// TwinCAT 3 PLC project PLC
// ProgramVersion: 3.1.4026.21
// libraries:
//   mobject-core, * (mobject)
//   Tc2_Standard, * (Beckhoff Automation GmbH)
//   Tc2_System, * (Beckhoff Automation GmbH)
//   Tc2_Utilities, * (Beckhoff Automation GmbH)
// project tree:
//   EL2574/DUT/ EL2574_IO.TcDUT, EL2574_Command.TcDUT, EL2574_IO_Control_Color.TcDUT, EL2574_IO_Status.TcDUT, EL2574_IO_Control.TcDUT
//   EL2574/ EL2574_CommandMode.TcPOU, HtmlColorCodeToRGBA.TcPOU, Section.TcDUT
//   EL2574/Interface/ I_EL2574_CommandMode.TcIO
//   / MAIN.TcPOU, PlcTask.TcTTO
// real-time tasks:
//   TASK PlcTask: cycle T#10ms, priority 20, ADS port 350
// I/O:
//   DEVICE CX (EtherCAT), AmsNetId 0.0.0.0.2.1
//     Term 1 (EK1200) [EK1200-5000 EtherCAT Power supply (2A E-Bus)]
//       LED 1-4 (EL2574) [EL2574 4 Ch. Pixel LED Controller]
//         modules: SlotGroup 1 (Slot 1, 2) (2xASYNC), SlotGroup 1 (Slot 1, 2) (2xASYNC), SlotGroup 2 (Slot 3, 4) (2xASYNC), SlotGroup 2 (Slot 3, 4) (2xASYNC)
//       LED 5-8 (EL2574) [EL2574 4 Ch. Pixel LED Controller]
//         modules: SlotGroup 1 (Slot 1, 2) (2xASYNC), SlotGroup 1 (Slot 1, 2) (2xASYNC), SlotGroup 2 (Slot 3, 4) (2xASYNC), SlotGroup 2 (Slot 3, 4) (2xASYNC)
// variable links:
//   (this object) <-> CX (EtherCAT)/Term 1 (EK1200)/LED 1-4 (EL2574)
//     PlcTask Inputs/MAIN.LED1.pdo.Status <-> SlotGroup 1 (Slot 1, 2) (2xASYNC)/Status Channel 1/Status
//     PlcTask Inputs/MAIN.LED2.pdo.Status <-> SlotGroup 1 (Slot 1, 2) (2xASYNC)/Status Channel 2/Status
//     PlcTask Inputs/MAIN.LED3.pdo.Status <-> SlotGroup 2 (Slot 3, 4) (2xASYNC)/Status Channel 1/Status
//     PlcTask Inputs/MAIN.LED4.pdo.Status <-> SlotGroup 2 (Slot 3, 4) (2xASYNC)/Status Channel 2/Status
//     PlcTask Outputs/MAIN.LED1.pdo.Control <-> SlotGroup 1 (Slot 1, 2) (2xASYNC)/Control Channel 1/Control
//     PlcTask Outputs/MAIN.LED2.pdo.Control <-> SlotGroup 1 (Slot 1, 2) (2xASYNC)/Control Channel 2/Control
//     PlcTask Outputs/MAIN.LED3.pdo.Control <-> SlotGroup 2 (Slot 3, 4) (2xASYNC)/Control Channel 1/Control
//     PlcTask Outputs/MAIN.LED4.pdo.Control <-> SlotGroup 2 (Slot 3, 4) (2xASYNC)/Control Channel 2/Control
//   (this object) <-> CX (EtherCAT)/Term 1 (EK1200)/LED 5-8 (EL2574)
//     PlcTask Inputs/MAIN.LED5.pdo.Status <-> SlotGroup 1 (Slot 1, 2) (2xASYNC)/Status Channel 1/Status
//     PlcTask Outputs/MAIN.LED5.pdo.Control <-> SlotGroup 1 (Slot 1, 2) (2xASYNC)/Control Channel 1/Control

CONFIGURATION PLC
    RESOURCE PLC ON TwinCAT3
        TASK PlcTask(INTERVAL := T#10ms, PRIORITY := 20);
        PROGRAM MAIN WITH PlcTask : MAIN;
    END_RESOURCE
END_CONFIGURATION

// ---- EL2574/DUT/EL2574_IO.TcDUT
TYPE EL2574_IO :
	STRUCT
		Status	AT %I* : EL2574_IO_Status;
		Control AT %Q* : EL2574_IO_Control;
	END_STRUCT
END_TYPE

// ---- EL2574/DUT/EL2574_Command.TcDUT
TYPE EL2574_Command :
	STRUCT
		Send	   : BOOL;
		Update	   : BOOL;
		Command	   : USINT;
		Index	   : UINT;
		Length	   : UINT;
		Parameter  : UINT;
		ColorRed   : USINT;
		ColorGreen : USINT;
		ColorBlue  : USINT;
		ColorWhite : USINT;
	END_STRUCT
END_TYPE

// ---- EL2574/DUT/EL2574_IO_Control_Color.TcDUT
TYPE EL2574_IO_Control_Color :
	STRUCT
		Red	  : USINT;
		Green : USINT;
		Blue  : USINT;
		White : USINT;
	END_STRUCT
END_TYPE

// ---- EL2574/DUT/EL2574_IO_Status.TcDUT
TYPE EL2574_IO_Status :
	STRUCT
		Busy					 : BIT;
		Transmit				 : BIT;
		Send_Acknowledge		 : BIT;
		Update_Acknowledge		 : BIT;
		Command_Acknowledge		 : BIT;
		Command_Reject			 : BIT;
		Warning					 : BIT;
		Error					 : BIT;
		Input_Cycle_Counter_Bit0 : BIT;
		Input_Cycle_Counter_Bit1 : BIT;
        {attribute 'hide'}
		_reserved1				 : BIT;
        {attribute 'hide'}
		_reserved2				 : BIT;
        {attribute 'hide'}
		_reserved3				 : BIT;
        {attribute 'hide'}
		_reserved4				 : BIT;
        {attribute 'hide'}
		_reserved5				 : BIT;
        {attribute 'hide'}
		_reserved6				 : BIT;
	END_STRUCT
END_TYPE

// ---- EL2574/DUT/EL2574_IO_Control.TcDUT
TYPE EL2574_IO_Control :
	STRUCT
		Execute : BIT;
		Send	: BIT;
		Update	: BIT;
		{attribute 'hide'}
		_reserved1 : BIT;
		{attribute 'hide'}
		_reserved2 : BIT;
		{attribute 'hide'}
		_reserved3 : BIT;
		{attribute 'hide'}
		_reserved4 : BIT;
		{attribute 'hide'}
		_reserved5 : BIT;
		Command	   : USINT;
		Index	   : UINT;
		Length	   : UINT;
		Parameter  : UINT;
		Color	   : EL2574_IO_Control_Color;
	END_STRUCT
END_TYPE

// ---- EL2574/Section.TcDUT
{attribute 'qualified_only'}
{attribute 'strict'}
{attribute 'to_string'}
TYPE Section : (
		None := 0,
		Accelerometer,
		Drives,
		Converter,
		Linux,
		Safety
	);
END_TYPE

// ---- EL2574/Interface/I_EL2574_CommandMode.TcIO
INTERFACE I_EL2574_CommandMode

METHOD PUBLIC ClearAll : I_EL2574_CommandMode
VAR_INPUT
END_VAR
END_METHOD

METHOD PUBLIC ColorGradient2Point : I_EL2574_CommandMode
VAR_INPUT
	StartPosition  : UINT;
	NumberOfPixels : UINT;
	Color1		   : STRING(9);
	Color2		   : STRING(9);
END_VAR
END_METHOD

METHOD PUBLIC ColorGradient3Point : I_EL2574_CommandMode
VAR_INPUT
	StartPosition  : UINT;
	NumberOfPixels : UINT;
	Color1		   : STRING(9);
	Color2		   : STRING(9);
	Color3		   : STRING(9);
END_VAR
END_METHOD

METHOD PUBLIC ColorGradient4Point : I_EL2574_CommandMode
VAR_INPUT
	StartPosition  : UINT;
	NumberOfPixels : UINT;
	Color1		   : STRING(9);
	Color2		   : STRING(9);
	Color3		   : STRING(9);
	Color4		   : STRING(9);
END_VAR
END_METHOD

METHOD PUBLIC CopyPixels : I_EL2574_CommandMode
VAR_INPUT
	StartPosition  : UINT;
	NumberOfPixels : UINT;
	TargetPosition : UINT;
END_VAR
END_METHOD

METHOD PUBLIC FillColor : I_EL2574_CommandMode
VAR_INPUT
	StartPosition  : UINT;
	NumberOfPixels : UINT;
	Red			   : USINT;
	Green		   : USINT;
	Blue		   : USINT;
	White		   : USINT;
END_VAR
END_METHOD

METHOD PUBLIC Invert : I_EL2574_CommandMode
VAR_INPUT
	StartPosition  : UINT;
	NumberOfPixels : UINT;
END_VAR
END_METHOD

METHOD PUBLIC MovePixels : I_EL2574_CommandMode
VAR_INPUT
	StartPosition  : UINT;
	NumberOfPixels : UINT;
	TargetPosition : UINT;
END_VAR
END_METHOD

METHOD PUBLIC RotateLeft : I_EL2574_CommandMode
VAR_INPUT
	StartPosition  : UINT;
	NumberOfPixels : UINT;
	Shift		   : UINT;
END_VAR
END_METHOD

METHOD PUBLIC RotateRight : I_EL2574_CommandMode
VAR_INPUT
	StartPosition  : UINT;
	NumberOfPixels : UINT;
	Shift		   : UINT;
END_VAR
END_METHOD

METHOD PUBLIC Send : I_EL2574_CommandMode
VAR_INPUT
END_VAR
END_METHOD

METHOD PUBLIC SendAndUpdate : I_EL2574_CommandMode
VAR_INPUT
END_VAR
END_METHOD

METHOD PUBLIC Update : I_EL2574_CommandMode
VAR_INPUT
END_VAR
END_METHOD

END_INTERFACE

// ---- MAIN.TcPOU
PROGRAM MAIN
VAR
	BackgroundColor		   : STRING(9) := '#fffafa';
	BackgroundColorRGB	   : ARRAY[0..3] OF USINT;
	DisplaySection		   : Section := Section.Linux;
	LED1				   : EL2574_CommandMode(10);
	LED2				   : EL2574_CommandMode(10);
	LED3				   : EL2574_CommandMode(10);
	LED4				   : EL2574_CommandMode(10);
	LED5				   : EL2574_CommandMode(10);
	onChange			   : r_Trig;
	previousDisplaySection : Section;
	State				   : (Idle,
		Clear,
		SetColor,
		SetColorUpdate);
	UpdateTon : TON;
	start	  : UINT;
	end		  : UINT;
END_VAR

VAR CONSTANT
	WHITE  : ARRAY[0..2] OF USINT := [255, 255, 255];
	RED	   : ARRAY[0..2] OF USINT := [255, 0, 0];
	BLUE   : ARRAY[0..2] OF USINT := [0, 0, 255];
	GREEN  : ARRAY[0..2] OF USINT := [0, 255, 0];
	YELLOW : ARRAY[0..2] OF USINT := [255, 255, 0];
END_VAR

BackgroundColorRGB := HtmlColorCodeToRGBA(BackgroundColor);
CASE State OF
	Idle:
		onChange(CLK := previousDisplaySection <> DisplaySection);
		IF OnChange.Q THEN
			PreviousDisplaySection := DisplaySection;
			LED1.ClearAll();
			LED2.ClearAll();
			LED3.ClearAll();
			LED4.FillColor(0,
						   75,
						   BackgroundColorRGB[0],
						   BackgroundColorRGB[1],
						   BackgroundColorRGB[2],
						   0);

			LED5.FillColor(0,
						   75,
						   BackgroundColorRGB[0],
						   BackgroundColorRGB[1],
						   BackgroundColorRGB[2],
						   0);

			State := Clear;
		END_IF

	Clear:
		UpdateTon(IN := TRUE, PT := T#100MS);
		IF UpdateTon.Q THEN
			UpdateTon(IN := FALSE);
			LED1.Update();
			LED2.Update();
			LED3.Update();
			LED4.Update();
			LED5.Update();
			State := SetColor;
		END_IF

	SetColor:
		CASE DisplaySection OF
			Section.None:
			Section.Accelerometer:
				LED2.FillColor(3,
							   3,
							   GREEN[0],
							   GREEN[1],
							   GREEN[2],
							   0);

			Section.Drives:
				LED1.FillColor(0,
							   100,
							   RED[0],
							   RED[1],
							   RED[2],
							   0);

				LED2.FillColor(0,
							   2,
							   RED[0],
							   RED[1],
							   RED[2],
							   0);

				LED3.ClearAll();

			Section.Linux:
				LED2.FillColor(4,
							   5,
							   WHITE[0],
							   WHITE[1],
							   WHITE[2],
							   0);

				LED3.ClearAll();

			Section.Safety:
				LED1.FillColor(0,
							   100,
							   YELLOW[0],
							   YELLOW[1],
							   YELLOW[2],
							   0);

				LED2.FillColor(0,
							   2,
							   YELLOW[0],
							   YELLOW[1],
							   YELLOW[2],
							   0);

				LED3.FillColor(0,
							   100,
							   YELLOW[0],
							   YELLOW[1],
							   YELLOW[2],
							   0);

			Section.Converter:
				LED2.FillColor(0,
							   2,
							   0,
							   0,
							   0,
							   0);

				LED2.FillColor(3,
							   3,
							   BLUE[0],
							   BLUE[1],
							   BLUE[2],
							   0);

				LED2.FillColor(4,
							   5,
							   0,
							   0,
							   0,
							   0);
		END_CASE

		State := SetColorUpdate;

	SetColorUpdate:
		UpdateTon(IN := TRUE, PT := T#100MS);
		IF UpdateTon.Q THEN
			UpdateTon(IN := FALSE);
			LED1.Update();
			LED2.Update();
			LED3.Update();
			LED4.Update();
			LED5.Update();
			State := IDLE;
		END_IF
END_CASE

LED1.CyclicCall();
LED2.CyclicCall();
LED3.CyclicCall();
LED4.CyclicCall();
LED5.CyclicCall();

END_PROGRAM

// ---- EL2574/EL2574_CommandMode.TcPOU
FUNCTION_BLOCK EL2574_CommandMode IMPLEMENTS I_EL2574_CommandMode
VAR
	totalPixels : UDINT;
	pdo			: EL2574_IO;
	commands	: Queue;
	errored		: BOOL;
END_VAR

VAR CONSTANT
	MAX_PIXELS			   : UDINT := 2048;
	COMMAND_NOP			   : USINT := 16#00;
	COMMAND_FILL		   : USINT := 16#01;
	COMMAND_CLEAR		   : USINT := 16#02;
	COMMAND_COPY		   : USINT := 16#03;
	COMMAND_MOVE		   : USINT := 16#04;
	COMMAND_ROTATE_LEFT	   : USINT := 16#05;
	COMMAND_ROTATE_RIGHT   : USINT := 16#06;
	COMMAND_REVERSE		   : USINT := 16#07;
	COMMAND_GRADIENT_START : USINT := 16#08;
	COMMAND_GRADIENT_END   : USINT := 16#09;
END_VAR

METHOD PUBLIC ClearAll : I_EL2574_CommandMode
VAR_INPUT
END_VAR

VAR
	command : EL2574_Command;
END_VAR
command.Send	   := FALSE;
command.Update	   := FALSE;
command.Command	   := COMMAND_CLEAR;
command.Index	   := 0;
command.Length	   := 0;
command.Parameter  := 0;
command.ColorRed   := 0;
command.ColorGreen := 0;
command.ColorBlue  := 0;
command.ColorWhite := 0;
commands.Enqueue(command);
ClearAll := THIS^;
END_METHOD

METHOD PUBLIC ColorGradient2Point : I_EL2574_CommandMode
VAR_INPUT
	StartPosition  : UINT;
	NumberOfPixels : UINT;
	Color1		   : STRING(9);
	Color2		   : STRING(9);
END_VAR
EnqueueGradientStart(StartPosition, NumberOfPixels, Color1);
EnqueueGradientEnd(StartPosition, NumberOfPixels, Color2);
ColorGradient2Point := THIS^;
END_METHOD

METHOD PUBLIC ColorGradient3Point : I_EL2574_CommandMode
VAR_INPUT
	StartPosition  : UINT;
	NumberOfPixels : UINT;
	Color1		   : STRING(9);
	Color2		   : STRING(9);
	Color3		   : STRING(9);
END_VAR

VAR
	segmentSize		 : UINT;
	finalSegmentSize : UINT;
	midpointStart	 : UINT;
END_VAR
IF NumberOfPixels < 3 THEN
	RETURN;
END_IF

segmentSize		 := NumberOfPixels / 2;
finalSegmentSize := NumberOfPixels - segmentSize;
midpointStart	 := StartPosition + segmentSize;
EnqueueGradientStart(StartPosition, segmentSize, Color1);
EnqueueGradientEnd(StartPosition, segmentSize, Color2);
EnqueueGradientStart(midpointStart, finalSegmentSize, Color2);
EnqueueGradientEnd(midpointStart, finalSegmentSize, Color3);
ColorGradient3Point := THIS^;
END_METHOD

METHOD PUBLIC ColorGradient4Point : I_EL2574_CommandMode
VAR_INPUT
	StartPosition  : UINT;
	NumberOfPixels : UINT;
	Color1		   : STRING(9);
	Color2		   : STRING(9);
	Color3		   : STRING(9);
	Color4		   : STRING(9);
END_VAR

VAR
	segmentSize		 : UINT;
	finalSegmentSize : UINT;
	firstThirdStart	 : UINT;
	secondThirdStart : UINT;
END_VAR
IF NumberOfPixels < 3 THEN
	RETURN;
END_IF

segmentSize		 := NumberOfPixels / 3;
firstThirdStart	 := StartPosition + segmentSize;
secondThirdStart := StartPosition + segmentSize * 2;
finalSegmentSize := NumberOfPixels - (segmentSize * 2);
EnqueueGradientStart(StartPosition, segmentSize, Color1);
EnqueueGradientEnd(StartPosition, segmentSize, Color2);
EnqueueGradientStart(firstThirdStart, segmentSize, Color2);
EnqueueGradientEnd(firstThirdStart, segmentSize, Color3);
EnqueueGradientStart(secondThirdStart, finalSegmentSize, Color3);
EnqueueGradientEnd(secondThirdStart, finalSegmentSize, Color4);
ColorGradient4Point := THIS^;
END_METHOD

METHOD PUBLIC CopyPixels : I_EL2574_CommandMode
VAR_INPUT
	StartPosition  : UINT;
	NumberOfPixels : UINT;
	TargetPosition : UINT;
END_VAR

VAR
	command : EL2574_Command;
END_VAR
command.Send	   := FALSE;
command.Update	   := FALSE;
command.Command	   := COMMAND_COPY;
command.Index	   := StartPosition;
command.Length	   := NumberOfPixels;
command.Parameter  := TargetPosition;
command.ColorRed   := 0;
command.ColorGreen := 0;
command.ColorBlue  := 0;
command.ColorWhite := 0;
commands.Enqueue(command);
CopyPixels := THIS^;
END_METHOD

METHOD PUBLIC CyclicCall
VAR_INPUT
END_VAR

VAR
	sendCommand : EL2574_Command;
END_VAR
IF pdo.Status.Busy THEN
	RETURN;
END_IF

IF pdo.Status.Transmit THEN
	RETURN;
END_IF

IF commands.IsEmpty THEN
	RETURN;
END_IF

IF NOT commands.TryDequeue(sendCommand) THEN
	errored := TRUE;
	RETURN;
END_IF

pdo.Control.Send		:= sendCommand.Send;
pdo.Control.Update		:= sendCommand.Update;
pdo.Control.Command		:= sendCommand.Command;
pdo.Control.Index		:= sendCommand.Index;
pdo.Control.Length		:= sendCommand.Length;
pdo.Control.Parameter	:= sendCommand.Parameter;
pdo.Control.Color.Red	:= sendCommand.ColorRed;
pdo.Control.Color.Green := sendCommand.ColorGreen;
pdo.Control.Color.Blue	:= sendCommand.ColorBlue;
pdo.Control.Color.White := sendCommand.ColorWhite;
pdo.Control.Execute		:= NOT pdo.Control.Execute;
END_METHOD

METHOD PRIVATE EnqueueGradientEnd
VAR_INPUT
	StartPosition  : UINT;
	NumberOfPixels : UINT;
	Color		   : STRING(9);
END_VAR

VAR
	convertedColor : ARRAY[0..3] OF USINT;
	command		   : EL2574_Command;
END_VAR
convertedColor	   := HtmlColorCodeToRGBA(Color);
command.Send	   := FALSE;
command.Update	   := FALSE;
command.Command	   := COMMAND_GRADIENT_END;
command.Index	   := StartPosition;
command.Length	   := NumberOfPixels;
command.Parameter  := 0;
command.ColorRed   := convertedColor[0];
command.ColorGreen := convertedColor[1];
command.ColorBlue  := convertedColor[2];
command.ColorWhite := convertedColor[3];
commands.Enqueue(command);
END_METHOD

METHOD PRIVATE EnqueueGradientStart
VAR_INPUT
	StartPosition  : UINT;
	NumberOfPixels : UINT;
	Color		   : STRING(9);
END_VAR

VAR
	convertedColor : ARRAY[0..3] OF USINT;
	command		   : EL2574_Command;
END_VAR
convertedColor	   := HtmlColorCodeToRGBA(Color);
command.Send	   := FALSE;
command.Update	   := FALSE;
command.Command	   := COMMAND_GRADIENT_START;
command.Index	   := StartPosition;
command.Length	   := NumberOfPixels;
command.Parameter  := 0;
command.ColorRed   := convertedColor[0];
command.ColorGreen := convertedColor[1];
command.ColorBlue  := convertedColor[2];
command.ColorWhite := convertedColor[3];
commands.Enqueue(command);
END_METHOD

METHOD FB_init : BOOL
VAR_INPUT
	bInitRetains : BOOL; // if TRUE, the retain variables are initialized (warm start / cold start)
	bInCopyCode	 : BOOL; // if TRUE, the instance afterwards gets moved into the copy code (online change)
	TotalPixels	 : UDINT;
END_VAR
THIS^.totalPixels := TotalPixels;
END_METHOD

METHOD PUBLIC FillColor : I_EL2574_CommandMode
VAR_INPUT
	StartPosition  : UINT;
	NumberOfPixels : UINT;
	Red			   : USINT;
	Green		   : USINT;
	Blue		   : USINT;
	White		   : USINT;
END_VAR

VAR
	command : EL2574_Command;
END_VAR
command.Send	   := FALSE;
command.Update	   := FALSE;
command.Command	   := COMMAND_FILL;
command.Index	   := StartPosition;
command.Length	   := NumberOfPixels;
command.Parameter  := 0;
command.ColorRed   := Red;
command.ColorGreen := Green;
command.ColorBlue  := Blue;
command.ColorWhite := White;
commands.Enqueue(command);
FillColor := THIS^;
END_METHOD

PROPERTY PUBLIC HasError : BOOL
GET
HasError := errored;
END_GET
END_PROPERTY

METHOD PUBLIC Invert : I_EL2574_CommandMode
VAR_INPUT
	StartPosition  : UINT;
	NumberOfPixels : UINT;
END_VAR

VAR
	command : EL2574_Command;
END_VAR
command.Send	   := FALSE;
command.Update	   := FALSE;
command.Command	   := COMMAND_REVERSE;
command.Index	   := StartPosition;
command.Length	   := NumberOfPixels;
command.Parameter  := 0;
command.ColorRed   := 0;
command.ColorGreen := 0;
command.ColorBlue  := 0;
command.ColorWhite := 0;
commands.Enqueue(command);
Invert := THIS^;
END_METHOD

PROPERTY PUBLIC IsBusy : BOOL
GET
IsBusy := pdo.Status.Busy OR NOT commands.IsEmpty;
END_GET
END_PROPERTY

METHOD PUBLIC MovePixels : I_EL2574_CommandMode
VAR_INPUT
	StartPosition  : UINT;
	NumberOfPixels : UINT;
	TargetPosition : UINT;
END_VAR

VAR
	command : EL2574_Command;
END_VAR
command.Send	   := FALSE;
command.Update	   := FALSE;
command.Command	   := COMMAND_MOVE;
command.Index	   := StartPosition;
command.Length	   := NumberOfPixels;
command.Parameter  := TargetPosition;
command.ColorRed   := 0;
command.ColorGreen := 0;
command.ColorBlue  := 0;
command.ColorWhite := 0;
commands.Enqueue(command);
MovePixels := THIS^;
END_METHOD

METHOD PUBLIC RotateLeft : I_EL2574_CommandMode
VAR_INPUT
	StartPosition  : UINT;
	NumberOfPixels : UINT;
	Shift		   : UINT;
END_VAR

VAR
	command : EL2574_Command;
END_VAR
command.Send	   := FALSE;
command.Update	   := FALSE;
command.Command	   := COMMAND_ROTATE_LEFT;
command.Index	   := StartPosition;
command.Length	   := NumberOfPixels;
command.Parameter  := Shift;
command.ColorRed   := 0;
command.ColorGreen := 0;
command.ColorBlue  := 0;
command.ColorWhite := 0;
commands.Enqueue(command);
RotateLeft := THIS^;
END_METHOD

METHOD PUBLIC RotateRight : I_EL2574_CommandMode
VAR_INPUT
	StartPosition  : UINT;
	NumberOfPixels : UINT;
	Shift		   : UINT;
END_VAR

VAR
	command : EL2574_Command;
END_VAR
command.Send	   := FALSE;
command.Update	   := FALSE;
command.Command	   := COMMAND_ROTATE_RIGHT;
command.Index	   := StartPosition;
command.Length	   := NumberOfPixels;
command.Parameter  := Shift;
command.ColorRed   := 0;
command.ColorGreen := 0;
command.ColorBlue  := 0;
command.ColorWhite := 0;
commands.Enqueue(command);
RotateRight := THIS^;
END_METHOD

METHOD PUBLIC Send : I_EL2574_CommandMode
VAR_INPUT
END_VAR

VAR
	command : EL2574_Command;
END_VAR
command.Send	   := TRUE;
command.Update	   := FALSE;
command.Command	   := COMMAND_NOP;
command.Index	   := 0;
command.Length	   := 0;
command.Parameter  := 0;
command.ColorRed   := 0;
command.ColorGreen := 0;
command.ColorBlue  := 0;
command.ColorWhite := 0;
commands.Enqueue(command);
Send := THIS^;
END_METHOD

METHOD PUBLIC SendAndUpdate : I_EL2574_CommandMode
VAR_INPUT
END_VAR

VAR
	command : EL2574_Command;
END_VAR
command.Send	   := TRUE;
command.Update	   := TRUE;
command.Command	   := COMMAND_NOP;
command.Index	   := 0;
command.Length	   := 0;
command.Parameter  := 0;
command.ColorRed   := 0;
command.ColorGreen := 0;
command.ColorBlue  := 0;
command.ColorWhite := 0;
commands.Enqueue(command);
SendAndUpdate := THIS^;
END_METHOD

METHOD PUBLIC Update : I_EL2574_CommandMode
VAR_INPUT
END_VAR

VAR
	command : EL2574_Command;
END_VAR
command.Send	   := FALSE;
command.Update	   := TRUE;
command.Command	   := COMMAND_NOP;
command.Index	   := 0;
command.Length	   := 0;
command.Parameter  := 0;
command.ColorRed   := 0;
command.ColorGreen := 0;
command.ColorBlue  := 0;
command.ColorWhite := 0;
commands.Enqueue(command);
Update := THIS^;
END_METHOD

END_FUNCTION_BLOCK

// ---- EL2574/HtmlColorCodeToRGBA.TcPOU
FUNCTION HtmlColorCodeToRGBA : ARRAY [0..3] OF USINT
VAR_INPUT
	ColorCode : STRING(9);
END_VAR
VAR
	toConvert : STRING;
	converted : ARRAY [0..3] OF USINT;
END_VAR

// allow the user to pass in the # as optional
IF FIND(ColorCode,'#') = 1 THEN
	toConvert := right(ColorCode, len(ColorCode)-1);
ELSE
	toConvert := ColorCode;
END_IF

// check for a valid string, i.e. must be 6 or 8 chars long.
IF NOT(len(toConvert) = 6 OR len(toConvert) = 8) THEN
	RETURN;
END_IF

// allow 6 or 8 hex codes
IF len(toConvert) = 6 THEN
	toConvert := concat(toConvert,'00');
END_IF

HEXSTR_TO_DATA( toConvert, ADR(converted), SIZEOF(converted));
HtmlColorCodeToRGBA := converted;

END_FUNCTION
